// Retrieves the positive infinity value for LREAL data type.
FUNCTION F_GetInf : LREAL // The positive infinity value.
VAR_STAT
	fInf : LREAL := TO_LREAL('#Inf');
END_VAR

F_GetInf := fInf;

END_FUNCTION

(* stored: Version 1.1.0.1
   POU F_GetInf: Id {a54a29e2-7027-0a3f-10f3-ad3832c32c82}, SpecialFunc None *)
